RoboDK station: PintaPiezas_Dominguez_Ramirez.rdk

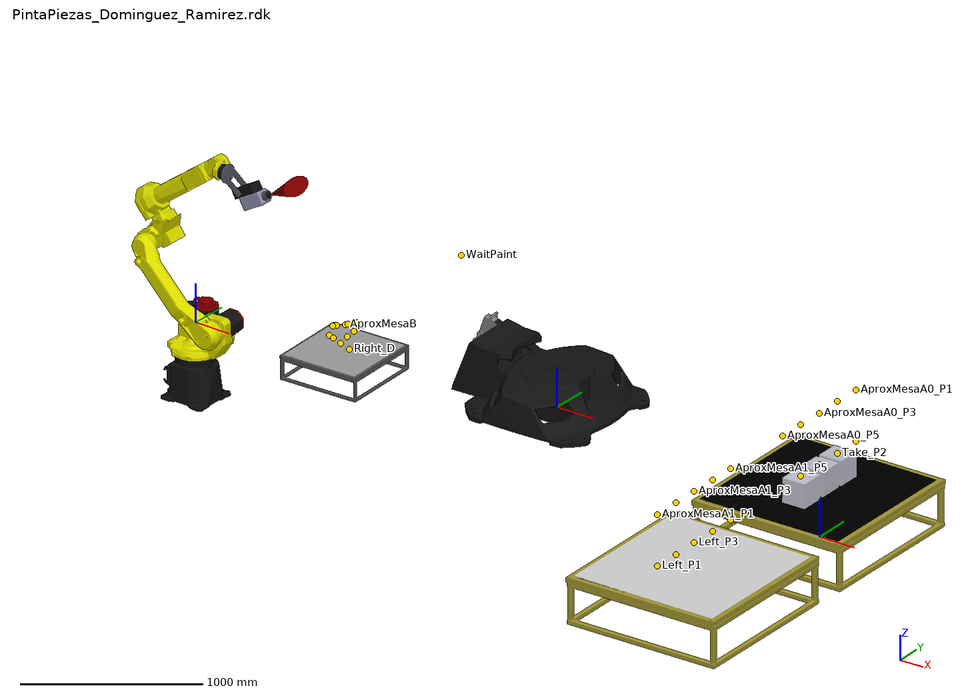
[picture v0: the station drawn from its stored meshes, robots at their saved joint values, targets as dots, program paths as lines]
Station PintaPiezas_Dominguez_Ramirez (saved by RoboDK 5.3.0). Poses are relative to the parent item; angles as X-Y-Z fixed-axis rotations.
Station parameters (name, value as stored): ColorObject, 3
  - Python program Preparar_Pieza1 (listed below)
  - Python program Pintar_Pieza1 (listed below)
  - Python program Almacenar_Pieza1 (listed below)
  - Python program Preparar_Pieza2 (listed below)
  - Python program Pintar_Pieza2 (listed below)
  - Python program Almacenar_Pieza2 (listed below)
  - Python program Preparar_Pieza3 (listed below)
  - Python program Pintar_Pieza3 (listed below)
  - Python program Almacenar_Pieza3 (listed below)
  - object MesaA at (3000, -2200, 0) mm, size 985.8 x 1004.9 x 291.9 mm, geometry from Table-108x114x32-IN.sld
    - object Pieza1 at (0, 1375, 429.65) mm, size 150 x 150 x 150 mm, geometry from box.sld
    - object Pieza2 at (0, 1200, 429.65) mm, size 150 x 150 x 150 mm, geometry from box.sld
    - object Pieza3 at (0, 1025, 429.65) mm, size 150 x 150 x 150 mm, geometry from box.sld
  - object MesaB at (0, 0, 0) mm, size 503 x 512.7 x 148.9 mm, geometry from Table-108x114x32-IN.sld
  - frame RobotA Base at (1676.97, -1606.48, 650) mm
    - robot RobotA (model KUKA KR 210 R2700 prime): 6 axes, payload 210 kg, reach 2696 mm, repeatability 0.06 mm, weight 1111 kg
        joint limits [-185, -140, -120, -350, -122.5, -350] to [185, -5, 155, 350, 122.5, 350]; home [0, -90, 90, 0, 0, 0]; saved at [-179.617, -136.253, 154.914, 0, 71.339, -179.617]
      - tool RobotiQ Sanding Kit, TCP at (0, 0, 90.86) mm, size 127 x 139.7 x 103.3 mm
    - target AproxMesaA0_P1 (Cartesian target) at (1323.03, 955.18, 93.07) mm, rotated rx 180 ry 0 rz 0 deg; joints [35.828, 52.673, -25.551, 0, -64.449, -35.828] of RobotA
    - target AproxMesaA0_P2 (Cartesian target) at (1323.03, 780.66, 93.07) mm, rotated rx 180 ry 0 rz 0 deg; joints [30.543, 46.178, -31.005, 0, -58.995, -30.543] of RobotA
    - target AproxMesaA0_P3 (Cartesian target) at (1323.03, 606.48, 93.07) mm, rotated rx -180 ry 0 rz 0 deg; joints [24.627, 41.286, -34.872, 0, -55.128, -24.627] of RobotA
    - target AproxMesaA0_P4 (Cartesian target) at (1323.03, 430.87, 93.07) mm, rotated rx -180 ry 0 rz 0 deg; joints [18.039, 37.651, -37.592, 0, -52.408, -18.039] of RobotA
    - target AproxMesaA0_P5 (Cartesian target) at (1323.03, 257.29, 93.07) mm, rotated rx -180 ry 0 rz 0 deg; joints [11.005, 35.26, -39.302, 0, -50.698, -11.005] of RobotA
    - target AproxMesaA1_P1 (Cartesian target) at (1323.03, -935.11, 93.07) mm, rotated rx -180 ry 0 rz 0 deg; joints [-35.252, 51.823, -26.284, 0, -63.716, 35.252] of RobotA
    - target AproxMesaA1_P2 (Cartesian target) at (1323.03, -761.53, 93.07) mm, rotated rx -180 ry 0 rz 0 deg; joints [-29.925, 45.572, -31.496, 0, -58.504, 29.925] of RobotA
    - target AproxMesaA1_P3 (Cartesian target) at (1323.03, -585.91, 93.07) mm, rotated rx -180 ry 0 rz 0 deg; joints [-23.886, 40.795, -35.247, 0, -54.753, 23.886] of RobotA
    - target AproxMesaA1_P4 (Cartesian target) at (1323.03, -411.74, 93.07) mm, rotated rx -180 ry 0 rz 0 deg; joints [-17.287, 37.329, -37.826, 0, -52.174, 17.287] of RobotA
    - target AproxMesaA1_P5 (Cartesian target) at (1323.03, -237.21, 93.07) mm, rotated rx -180 ry 0 rz 0 deg; joints [-10.165, 35.061, -39.441, 0, -50.559, 10.165] of RobotA
    - target Take_P1 (Cartesian target) at (1323.03, 956.48, -220.35) mm, rotated rx -180 ry 0 rz 0 deg; joints [35.865, 62.489, -38.726, 0, -51.274, -35.865] of RobotA
    - target Take_P2 (Cartesian target) at (1323.03, 780.66, -220.35) mm, rotated rx -180 ry 0 rz 0 deg; joints [30.543, 56.858, -44.792, 0, -45.208, -30.543] of RobotA
    - target Take_P3 (Cartesian target) at (1323.03, 606.48, -220.35) mm, rotated rx -180 ry 0 rz 0 deg; joints [24.627, 52.739, -49.29, 0, -40.71, -24.627] of RobotA
    - target Take_P4 (Cartesian target) at (1323.03, 430.87, -220.35) mm, rotated rx -180 ry 0 rz 0 deg; joints [18.039, 49.747, -52.598, 0, -37.402, -18.039] of RobotA
    - target Take_P5 (Cartesian target) at (1323.03, 257.29, -220.35) mm, rotated rx -180 ry 0 rz 0 deg; joints [11.005, 47.819, -54.753, 0, -35.247, -11.005] of RobotA
    - target Left_P1 (Cartesian target) at (1323.03, -933.81, -220.35) mm, rotated rx -180 ry 0 rz 0 deg; joints [-35.215, 61.659, -39.615, 0, -50.385, 35.215] of RobotA
    - target Left_P2 (Cartesian target) at (1323.03, -760.23, -220.35) mm, rotated rx -180 ry 0 rz 0 deg; joints [-29.882, 56.308, -45.389, 0, -44.611, 29.882] of RobotA
    - target Left_P3 (Cartesian target) at (1323.03, -584.61, -220.35) mm, rotated rx -180 ry 0 rz 0 deg; joints [-23.839, 52.306, -49.766, 0, -40.234, 23.839] of RobotA
    - target Left_P4 (Cartesian target) at (1323.03, -410.44, -220.35) mm, rotated rx -180 ry 0 rz 0 deg; joints [-17.235, 49.468, -52.909, 0, -37.091, 17.235] of RobotA
    - target Left_P5 (Cartesian target) at (1323.03, -235.91, -220.35) mm, rotated rx -180 ry 0 rz 0 deg; joints [-10.11, 47.649, -54.944, 0, -35.056, 10.11] of RobotA
    - target AproxMesaB (Cartesian target) at (-1417.07, 4.29, 103.23) mm, rotated rx 180 ry 0 rz 0 deg; joints [179.826, 38.777, -36.006, 0, -53.994, -179.826] of RobotA
    - target WaitPaint (Cartesian target) at (-643.02, 4.29, 741.53) mm, rotated rx 180 ry 0 rz 0 deg; joints [179.617, -20.046, -8.465, 0, -81.535, -179.617] of RobotA
    - frame MesaA0 Base at (1323.03, 606.48, -660.35) mm
      - object MesaC at (0, 0, 0) mm, size 985.8 x 1004.9 x 291.9 mm, geometry from Table-108x114x32-IN.sld
  - frame RobotB Base at (-785.52, -1535.25, 450) mm, rotated rx 0 ry 0 rz -3 deg
    - robot RobotB (model Fanuc M-10iA): 6 axes, payload 10 kg, reach 1420 mm, repeatability 0.08 mm, weight 130 kg
        modified DH rows (alpha deg, a mm, theta deg, d mm): 0, 0, 0, 450; -90, 150, -90, 0; 0, 600, 0, 0; -90, 200, 0, 640; 90, 0, 0, 0; -90, 0, 0, 100
        base shift (0, 0, -450) mm
        joint limits [-180, -90, -95, -190, -190, -360] to [180, 160, 180, 190, 190, 360]; home [0, -44.52, 36.95, 0, -36.95, 0]; saved at [0, -44.52, 36.95, 180, 36.95, 180]
      - tool Paint gun, TCP at (50, 0, 450) mm, rotated rx 0 ry 30 rz 0 deg, size 203.2 x 279.7 x 471.5 mm
    - target Right_D (Cartesian target) at (1128.46, -77.94, 203.78) mm, rotated rx 90 ry -60.18 rz -173.2 deg; joints [-28.769, 42.471, -20.584, -58.905, -97.457, 150.668] of RobotB
    - target Right_M (Cartesian target) at (1071.48, -84.74, 225.06) mm, rotated rx 90 ry -60.18 rz -173.2 deg; joints [-30.393, 36.873, -21.966, -58.048, -98.024, 152.655] of RobotB
    - target Right_U (Cartesian target) at (1002.27, -93, 254.88) mm, rotated rx 90 ry -60.18 rz -173.2 deg; joints [-32.542, 30.646, -22.514, -57, -99.408, 154.203] of RobotB
    - target Center_D (Cartesian target) at (1011.4, -39.87, 300.37) mm, rotated rx 180 ry 0 rz -173.2 deg; joints [-4.924, -0.5, 0.153, -6.683, -60.84, 193.459] of RobotB
    - target Center_M (Cartesian target) at (1050.89, 5.93, 300.37) mm, rotated rx 180 ry 0 rz -173.2 deg; joints [-1.501, 3.048, 0.227, -4.756, -60.572, 189.546] of RobotB
    - target Center_U (Cartesian target) at (1079.26, 49.09, 300.37) mm, rotated rx 180 ry 0 rz -173.2 deg; joints [1.46, 5.834, 0.429, -3.065, -60.572, 186.138] of RobotB
    - target Left_U (Cartesian target) at (1098.26, 69.52, 285.71) mm, rotated rx -90 ry 0 rz -173.2 deg; joints [33.722, 20.618, -41.647, 92.049, -87.698, 138.311] of RobotB
    - target Left_M (Cartesian target) at (1048.72, 63.61, 234.84) mm, rotated rx -90 ry 0 rz -173.2 deg; joints [35.116, 19.049, -47.063, 91.235, -88.851, 132.925] of RobotB
    - target Left_D (Cartesian target) at (1007.9, 58.74, 193.57) mm, rotated rx -90 ry 0 rz -173.2 deg; joints [36.368, 18.195, -51.506, 90.34, -89.729, 128.493] of RobotB
    - target Face_D (Cartesian target) at (972.74, -18.59, 202.79) mm, rotated rx 0 ry -90 rz -173.2 deg; joints [-9.324, -34.09, -22.694, 120.254, 16.17, 246.957] of RobotB
    - target Face_U (Cartesian target) at (973.71, -26.75, 277.71) mm, rotated rx 0 ry -90 rz -173.2 deg; joints [-10.259, -34.141, -16.259, 134.328, 20.806, 232.465] of RobotB
  - program MainProgram (9 instructions, listed below)

--- Python program Preparar_Pieza1 ---
from robolink import *    # RoboDK API
from robodk import *      # Robot toolBox
RDK = Robolink()

# Asignacion de objetos
toolA = 'RobotiQ Sanding Kit'
toolB = 'Paint gun'
objectA = 'Pieza1'
mesa1 = 'MesaB'
mesa2 = 'MesaA'
gripper1 = RDK.Item(toolA, ITEM_TYPE_TOOL)
gripper2 = RDK.Item(toolB, ITEM_TYPE_TOOL)
pi2 = RDK.Item(objectA, ITEM_TYPE_OBJECT)
mesapaint = RDK.Item(mesa1, ITEM_TYPE_OBJECT)
mesafinal = RDK.Item(mesa2, ITEM_TYPE_OBJECT)

# Configuracion RobotA
robotA = RDK.ItemUserPick('RobotA',ITEM_TYPE_ROBOT)
if not robotA.Valid():
    quit()
reference = robotA.Parent()
robotA.setPoseFrame(reference)
pose_ref = robotA.Pose()
print(Pose_2_TxyzRxyz(pose_ref))
home_joints = robotA.JointsHome().tolist()

# Preparar Pieza1 con Pick & Place

# RobotA se aproxima a MesaC para recoger la Pieza1
RDK.Spray_Clear()               # Se resetea el color de pintura
pi2.Recolor([0.90,0.91,0.96,1]) # Selecciona blanco como color inicial de la Pieza1
aprox=20
a1 = transl(1323.030,780.657,93.068)*roty(pi)
robotA.MoveJ(a1)
robotA.setSpeed(1000)

# RobotA toma la Pieza1 de la MesaC
b1 = transl(1323.030,780.657,-220.350)*roty(pi)
robotA.MoveJ(b1)
robotA.setSpeed(1000)
pi2.setParentStatic(gripper1)

# RobotA lleva la Pieza1 cerca de la MesaB
c1=transl(-1417.075,4.293,400.446)*roty(pi)
robotA.MoveJ(c1)
robotA.setSpeed(1000)

# RobotA deja la Pieza1 en la MesaB
d1=transl(-1417.075,4.293,100.367)*roty(pi)
robotA.MoveJ(d1)
robotA.setSpeed(1000)
gripper1.DetachAll()
pi2.setParentStatic(mesapaint)

# RobotA se ubica en la posición de espera
e1=transl(-643.019,4.293,741.529)*roty(pi)
robotA.MoveJ(e1)
robotA.setSpeed(1000)

--- Python program Pintar_Pieza1 ---
from robolink import *    # RoboDK API
from robodk import *      # Robot toolBox
RDK = Robolink()

# Asignacion de objetos
toolA = 'RobotiQ Sanding Kit'
toolB = 'Paint gun'
objectA = 'Pieza1'
mesa1 = 'MesaB'
mesa2 = 'MesaA'
gripper1 = RDK.Item(toolA, ITEM_TYPE_TOOL)
gripper2 = RDK.Item(toolB, ITEM_TYPE_TOOL)
pi1 = RDK.Item(objectA, ITEM_TYPE_OBJECT)
mesapaint = RDK.Item(mesa1, ITEM_TYPE_OBJECT)
mesafinal = RDK.Item(mesa2, ITEM_TYPE_OBJECT)

# Configuracion RobotB
robotB = RDK.ItemUserPick('RobotB',ITEM_TYPE_ROBOT)
if not robotB.Valid():
    quit()
reference1 = robotB.Parent()
robotB.setPoseFrame(reference1)
pose_ref1 = robotB.Pose()
print(Pose_2_TxyzRxyz(pose_ref1))
home_joints1 = robotB.JointsHome().tolist()

# RobotB pinta Pieza1
# Elegir color
color_object = 0
color_object_input = int(mbox('Seleccione un color ingresando el valor numerico correspondiente: 1=Rojo, 2=Verde, 3=Azul', entry=color_object))

# RobotB se aproxima a MesaB
aprox=20
a02 = xyzrpw_2_pose([951.091,-99.100,515.373,90.000,-60.175,-173.197])
robotB.MoveJ(a02)
robotB.setSpeed(100)

# Lado derecho
aprox=20
a2 = xyzrpw_2_pose([1128.463,-77.940,203.783,90.000,-60.175,-173.197])
robotB.MoveJ(a2)
robotB.setSpeed(100)
c2 = xyzrpw_2_pose([1071.476,-84.739,225.057,90.000,-60.175,-173.197])
robotB.MoveJ(c2)
robotB.setSpeed(1000)
d2 = xyzrpw_2_pose([1002.267,-92.996,254.878,90.000,-60.175,-173.197])
robotB.MoveJ(d2)
robotB.setSpeed(1000)

# Centro
e2 = xyzrpw_2_pose([1011.397,-39.866,300.368,180.000,0.000,-173.197])
robotB.MoveJ(e2)
robotB.setSpeed(1000)
f2 = xyzrpw_2_pose([1050.893,5.934,300.367,180.000,0.000,-173.197])
robotB.MoveJ(f2)
robotB.setSpeed(1000)
g2 = xyzrpw_2_pose([1079.262,49.092,300.367,180.000,0.000,-173.197])
robotB.MoveJ(g2)
robotB.setSpeed(1000)

# Lado izquierdo
h2 = xyzrpw_2_pose([1098.260,69.520,285.711,-90.000,0.000,-173.197])
robotB.MoveJ(h2)
robotB.setSpeed(1000)
i2 = xyzrpw_2_pose([1048.722,63.609,234.840,-90.000,0.000,-173.197])
robotB.MoveJ(i2)
robotB.setSpeed(1000)
j2 = xyzrpw_2_pose([1007.902,58.739,193.572,-90.000,0.000,-173.197])
robotB.MoveJ(j2)
robotB.setSpeed(1000)

# Frente
k2 = xyzrpw_2_pose([972.738,-18.594,202.789,0.000,-90.000,-173.197])
robotB.MoveJ(k2)
robotB.setSpeed(1000)
l2 = xyzrpw_2_pose([973.710,-26.748,277.710,0.000,-90.000,-173.197])
robotB.MoveJ(l2)
robotB.setSpeed(1000)

# Volver a la posicion inical
b2 = xyzrpw_2_pose([670.544,0.000,1022.351,0.000,-60.000,-180.000])
robotB.MoveJ(b2)
robotB.setSpeed(100)

# Color
if color_object_input == 1:
    pi1.Recolor([1,0,0,1])
elif color_object_input == 2:
    pi1.Recolor([0,1,0,1])
elif color_object_input == 3:
    pi1.Recolor([0,0,1,1])
else:
    pi1.Recolor([0.90,0.91,0.96,1])

--- Python program Almacenar_Pieza1 ---
from robolink import *    # RoboDK API
from robodk import *      # Robot toolBox
RDK = Robolink()

# Asignacion de objetos
toolA = 'RobotiQ Sanding Kit'
toolB = 'Paint gun'
objectA = 'Pieza1'
mesa1 = 'MesaB'
mesa2 = 'MesaA'
gripper1 = RDK.Item(toolA, ITEM_TYPE_TOOL)
gripper2 = RDK.Item(toolB, ITEM_TYPE_TOOL)
pi2 = RDK.Item(objectA, ITEM_TYPE_OBJECT)
mesapaint = RDK.Item(mesa2, ITEM_TYPE_OBJECT)
mesafinal = RDK.Item(mesa2, ITEM_TYPE_OBJECT)

# Configuracion RobotA
robotA = RDK.ItemUserPick('RobotA',ITEM_TYPE_ROBOT)
if not robotA.Valid():
    quit()
reference = robotA.Parent()
robotA.setPoseFrame(reference)
pose_ref = robotA.Pose()
print(Pose_2_TxyzRxyz(pose_ref))
home_joints = robotA.JointsHome().tolist()

# Almacenar Pieza1 con Pick & Place

# RobotA toma la Pieza1 de la MesaB
a3=transl(-1417.075,4.293,100.367)*roty(pi)
robotA.MoveJ(a3)
robotA.setSpeed(1000)
mesapaint.DetachAll()
pi2.setParentStatic(gripper1)

# RobotA lleva la Pieza1 lejos de la MesaB
b3=transl(-1417.075,4.293,400.446)*roty(pi)
robotA.MoveJ(b3)
robotA.setSpeed(1000)

# RobotA lleva la Pieza1 entre MesaB y MesaA
f3=transl(1323.030,780.657,93.068)*roty(pi)
robotA.MoveJ(f3)
robotA.setSpeed(1000)

# RobotA lleva la Pieza1 cerca de la MesaA
c3=transl(1323.030,-761.529,93.068)*roty(pi)
robotA.MoveJ(c3)
robotA.setSpeed(1000)

# RobotA deja la Pieza1 en la MesaA
d3=transl(1323.030,-760.228,-220.350)*roty(pi)
robotA.MoveJ(d3)
robotA.setSpeed(1000)
gripper1.DetachAll()
pi2.setParentStatic(mesafinal)

# Volver a la posicion inical
e3=transl(945.000,0.000,834.135)*roty(pi)
robotA.MoveJ(e3)
robotA.setSpeed(1000)

--- Python program Preparar_Pieza2 ---
from robolink import *    # RoboDK API
from robodk import *      # Robot toolBox
RDK = Robolink()

# Asignacion de objetos
toolA = 'RobotiQ Sanding Kit'
toolB = 'Paint gun'
objectB = 'Pieza2'
mesa1 = 'MesaB'
mesa2 = 'MesaA'
gripper1 = RDK.Item(toolA, ITEM_TYPE_TOOL)
gripper2 = RDK.Item(toolB, ITEM_TYPE_TOOL)
pi3 = RDK.Item(objectB, ITEM_TYPE_OBJECT)
mesapaint = RDK.Item(mesa1, ITEM_TYPE_OBJECT)
mesafinal = RDK.Item(mesa2, ITEM_TYPE_OBJECT)

# Configuracion RobotA
robotA = RDK.ItemUserPick('RobotA',ITEM_TYPE_ROBOT)
if not robotA.Valid():
    quit()
reference = robotA.Parent()
robotA.setPoseFrame(reference)
pose_ref = robotA.Pose()
print(Pose_2_TxyzRxyz(pose_ref))
home_joints = robotA.JointsHome().tolist()

# Preparar Pieza2 con Pick & Place

# RobotA se aproxima a MesaC para recoger la Pieza2
RDK.Spray_Clear()               # Se resetea el color de pintura
pi3.Recolor([0.90,0.91,0.96,1]) # Selecciona blanco como color inicial de la Pieza2
aprox=20
a1 = transl(1323.030,606.483,93.068)*roty(pi)
robotA.MoveJ(a1)
robotA.setSpeed(1000)

# RobotA toma la Pieza2 de la MesaC
b1 = transl(1323.030,606.483,-220.350)*roty(pi)
robotA.MoveJ(b1)
robotA.setSpeed(1000)
pi3.setParentStatic(gripper1)

# RobotA lleva la Pieza2 cerca de la MesaB
c1=transl(-1417.075,4.293,400.446)*roty(pi)
robotA.MoveJ(c1)
robotA.setSpeed(1000)

# RobotA deja la Pieza2 en la MesaB
d1=transl(-1417.075,4.293,100.367)*roty(pi)
robotA.MoveJ(d1)
robotA.setSpeed(1000)
gripper1.DetachAll()
pi3.setParentStatic(mesapaint)

# RobotA se ubica en la posición de espera
e1=transl(-643.019,4.293,741.529)*roty(pi)
robotA.MoveJ(e1)
robotA.setSpeed(1000)

--- Python program Pintar_Pieza2 ---
from robolink import *    # RoboDK API
from robodk import *      # Robot toolBox
RDK = Robolink()

# Asignacion de objetos
toolA = 'RobotiQ Sanding Kit'
toolB = 'Paint gun'
objectB = 'Pieza2'
mesa1 = 'MesaB'
mesa2 = 'MesaA'
gripper1 = RDK.Item(toolA, ITEM_TYPE_TOOL)
gripper2 = RDK.Item(toolB, ITEM_TYPE_TOOL)
pi2 = RDK.Item(objectB, ITEM_TYPE_OBJECT)
mesapaint = RDK.Item(mesa1, ITEM_TYPE_OBJECT)
mesafinal = RDK.Item(mesa2, ITEM_TYPE_OBJECT)

# Configuracion RobotB
robotB = RDK.ItemUserPick('RobotB',ITEM_TYPE_ROBOT)
if not robotB.Valid():
    quit()
reference1 = robotB.Parent()
robotB.setPoseFrame(reference1)
pose_ref1 = robotB.Pose()
print(Pose_2_TxyzRxyz(pose_ref1))
home_joints1 = robotB.JointsHome().tolist()

# RobotB pinta Pieza2
# Elegir color
color_object = 0
color_object_input = int(mbox('Seleccione un color ingresando el valor numerico correspondiente: 1=Rojo, 2=Verde, 3=Azul', entry=color_object))

# RobotB se aproxima a MesaB
aprox=20
a02 = xyzrpw_2_pose([951.091,-99.100,515.373,90.000,-60.175,-173.197])
robotB.MoveJ(a02)
robotB.setSpeed(100)

# Lado derecho
aprox=20
a2 = xyzrpw_2_pose([1128.463,-77.940,203.783,90.000,-60.175,-173.197])
robotB.MoveJ(a2)
robotB.setSpeed(100)
c2 = xyzrpw_2_pose([1071.476,-84.739,225.057,90.000,-60.175,-173.197])
robotB.MoveJ(c2)
robotB.setSpeed(1000)
d2 = xyzrpw_2_pose([1002.267,-92.996,254.878,90.000,-60.175,-173.197])
robotB.MoveJ(d2)
robotB.setSpeed(1000)

# Centro
e2 = xyzrpw_2_pose([1011.397,-39.866,300.368,180.000,0.000,-173.197])
robotB.MoveJ(e2)
robotB.setSpeed(1000)
f2 = xyzrpw_2_pose([1050.893,5.934,300.367,180.000,0.000,-173.197])
robotB.MoveJ(f2)
robotB.setSpeed(1000)
g2 = xyzrpw_2_pose([1079.262,49.092,300.367,180.000,0.000,-173.197])
robotB.MoveJ(g2)
robotB.setSpeed(1000)

# Lado izquierdo
h2 = xyzrpw_2_pose([1098.260,69.520,285.711,-90.000,0.000,-173.197])
robotB.MoveJ(h2)
robotB.setSpeed(1000)
i2 = xyzrpw_2_pose([1048.722,63.609,234.840,-90.000,0.000,-173.197])
robotB.MoveJ(i2)
robotB.setSpeed(1000)
j2 = xyzrpw_2_pose([1007.902,58.739,193.572,-90.000,0.000,-173.197])
robotB.MoveJ(j2)
robotB.setSpeed(1000)

# Frente
k2 = xyzrpw_2_pose([972.738,-18.594,202.789,0.000,-90.000,-173.197])
robotB.MoveJ(k2)
robotB.setSpeed(1000)
l2 = xyzrpw_2_pose([973.710,-26.748,277.710,0.000,-90.000,-173.197])
robotB.MoveJ(l2)
robotB.setSpeed(1000)

# Volver a la posicion inical
b2 = xyzrpw_2_pose([670.544,0.000,1022.351,0.000,-60.000,-180.000])
robotB.MoveJ(b2)
robotB.setSpeed(100)

#Color
if color_object_input == 1:
    pi2.Recolor([1,0,0,1])
elif color_object_input == 2:
    pi2.Recolor([0,1,0,1])
elif color_object_input == 3:
    pi2.Recolor([0,0,1,1])
else:
    pi2.Recolor([0.90,0.91,0.96,1])

--- Python program Almacenar_Pieza2 ---
from robolink import *    # RoboDK API
from robodk import *      # Robot toolBox
RDK = Robolink()

# Asignacion de objetos
toolA = 'RobotiQ Sanding Kit'
toolB = 'Paint gun'
objectB = 'Pieza2'
mesa1 = 'MesaB'
mesa2 = 'MesaA'
gripper1 = RDK.Item(toolA, ITEM_TYPE_TOOL)
gripper2 = RDK.Item(toolB, ITEM_TYPE_TOOL)
pi3 = RDK.Item(objectB, ITEM_TYPE_OBJECT)
mesapaint = RDK.Item(mesa2, ITEM_TYPE_OBJECT)
mesafinal = RDK.Item(mesa2, ITEM_TYPE_OBJECT)

# Configuracion RobotA
robotA = RDK.ItemUserPick('RobotA',ITEM_TYPE_ROBOT)
if not robotA.Valid():
    quit()
reference = robotA.Parent()
robotA.setPoseFrame(reference)
pose_ref = robotA.Pose()
print(Pose_2_TxyzRxyz(pose_ref))
home_joints = robotA.JointsHome().tolist()

# Almacenar Pieza2 con Pick & Place

# RobotA toma la Pieza2 de la MesaB
a3=transl(-1417.075,4.293,100.367)*roty(pi)
robotA.MoveJ(a3)
robotA.setSpeed(1000)
mesapaint.DetachAll()
pi3.setParentStatic(gripper1)

# RobotA lleva la Pieza2 lejos de la MesaB
b3=transl(-1417.075,4.293,400.446)*roty(pi)
robotA.MoveJ(b3)
robotA.setSpeed(1000)

# RobotA lleva la Pieza2 entre MesaB y MesaA
f3=transl(1323.030,606.483,93.068)*roty(pi)
robotA.MoveJ(f3)
robotA.setSpeed(1000)

# RobotA lleva la Pieza2 cerca de la MesaA
c3=transl(1323.030,-585.913,93.068)*roty(pi)
robotA.MoveJ(c3)
robotA.setSpeed(1000)

# RobotA deja la Pieza2 en la MesaA
d3=transl(1323.030,-584.612,-220.350)*roty(pi)
robotA.MoveJ(d3)
robotA.setSpeed(1000)
gripper1.DetachAll()
pi3.setParentStatic(mesafinal)

# Volver a la posicion inical
e3=transl(945.000,0.000,834.135)*roty(pi)
robotA.MoveJ(e3)
robotA.setSpeed(1000)

--- Python program Preparar_Pieza3 ---
from robolink import *    # RoboDK API
from robodk import *      # Robot toolBox
RDK = Robolink()

# Asignacion de objetos
toolA = 'RobotiQ Sanding Kit'
toolB = 'Paint gun'
objectC = 'Pieza3'
mesa1 = 'MesaB'
mesa2 = 'MesaA'
gripper1 = RDK.Item(toolA, ITEM_TYPE_TOOL)
gripper2 = RDK.Item(toolB, ITEM_TYPE_TOOL)
pi4 = RDK.Item(objectC, ITEM_TYPE_OBJECT)
mesapaint = RDK.Item(mesa1, ITEM_TYPE_OBJECT)
mesafinal = RDK.Item(mesa2, ITEM_TYPE_OBJECT)

# Configuracion RobotA
robotA = RDK.ItemUserPick('RobotA',ITEM_TYPE_ROBOT)
if not robotA.Valid():
    quit()
reference = robotA.Parent()
robotA.setPoseFrame(reference)
pose_ref = robotA.Pose()
print(Pose_2_TxyzRxyz(pose_ref))
home_joints = robotA.JointsHome().tolist()

# Preparar Pieza3 con Pick & Place

# RobotA se aproxima a MesaC para recoger la Pieza3
RDK.Spray_Clear()               # Se resetea el color de pintura
pi4.Recolor([0.90,0.91,0.96,1]) # Selecciona blanco como color inicial de la Pieza3
aprox=20
a1 = transl(1323.030,430.867,93.068)*roty(pi)
robotA.MoveJ(a1)
robotA.setSpeed(1000)

# RobotA toma la Pieza3 de la MesaC
b1 = transl(1323.030,430.867,-220.350)*roty(pi)
robotA.MoveJ(b1)
robotA.setSpeed(1000)
pi4.setParentStatic(gripper1)

# RobotA lleva la Pieza3 cerca de la MesaB
c1=transl(-1417.075,4.293,400.446)*roty(pi)
robotA.MoveJ(c1)
robotA.setSpeed(1000)

# RobotA deja la Pieza3 en la MesaB
d1=transl(-1417.075,4.293,100.367)*roty(pi)
robotA.MoveJ(d1)
robotA.setSpeed(1000)
gripper1.DetachAll()
pi4.setParentStatic(mesapaint)

# RobotA se ubica en la posición de espera
e1=transl(-643.019,4.293,741.529)*roty(pi)
robotA.MoveJ(e1)
robotA.setSpeed(1000)

--- Python program Pintar_Pieza3 ---
from robolink import *    # RoboDK API
from robodk import *      # Robot toolBox
RDK = Robolink()

# Asignacion de objetos
toolA = 'RobotiQ Sanding Kit'
toolB = 'Paint gun'
objectC = 'Pieza3'
mesa1 = 'MesaB'
mesa2 = 'MesaA'
gripper1 = RDK.Item(toolA, ITEM_TYPE_TOOL)
gripper2 = RDK.Item(toolB, ITEM_TYPE_TOOL)
pi3 = RDK.Item(objectC, ITEM_TYPE_OBJECT)
mesapaint = RDK.Item(mesa1, ITEM_TYPE_OBJECT)
mesafinal = RDK.Item(mesa2, ITEM_TYPE_OBJECT)

# Configuracion RobotB
robotB = RDK.ItemUserPick('RobotB',ITEM_TYPE_ROBOT)
if not robotB.Valid():
    quit()
reference1 = robotB.Parent()
robotB.setPoseFrame(reference1)
pose_ref1 = robotB.Pose()
print(Pose_2_TxyzRxyz(pose_ref1))
home_joints1 = robotB.JointsHome().tolist()

# RobotB pinta Pieza3
# Elegir color
color_object = 0
color_object_input = int(mbox('Seleccione un color ingresando el valor numerico correspondiente: 1=Rojo, 2=Verde, 3=Azul', entry=color_object))

# RobotB se aproxima a MesaB
aprox=20
a02 = xyzrpw_2_pose([951.091,-99.100,515.373,90.000,-60.175,-173.197])
robotB.MoveJ(a02)
robotB.setSpeed(100)

# Lado derecho
aprox=20
a2 = xyzrpw_2_pose([1128.463,-77.940,203.783,90.000,-60.175,-173.197])
robotB.MoveJ(a2)
robotB.setSpeed(100)
c2 = xyzrpw_2_pose([1071.476,-84.739,225.057,90.000,-60.175,-173.197])
robotB.MoveJ(c2)
robotB.setSpeed(1000)
d2 = xyzrpw_2_pose([1002.267,-92.996,254.878,90.000,-60.175,-173.197])
robotB.MoveJ(d2)
robotB.setSpeed(1000)

# Centro
e2 = xyzrpw_2_pose([1011.397,-39.866,300.368,180.000,0.000,-173.197])
robotB.MoveJ(e2)
robotB.setSpeed(1000)
f2 = xyzrpw_2_pose([1050.893,5.934,300.367,180.000,0.000,-173.197])
robotB.MoveJ(f2)
robotB.setSpeed(1000)
g2 = xyzrpw_2_pose([1079.262,49.092,300.367,180.000,0.000,-173.197])
robotB.MoveJ(g2)
robotB.setSpeed(1000)

# Lado izquierdo
h2 = xyzrpw_2_pose([1098.260,69.520,285.711,-90.000,0.000,-173.197])
robotB.MoveJ(h2)
robotB.setSpeed(1000)
i2 = xyzrpw_2_pose([1048.722,63.609,234.840,-90.000,0.000,-173.197])
robotB.MoveJ(i2)
robotB.setSpeed(1000)
j2 = xyzrpw_2_pose([1007.902,58.739,193.572,-90.000,0.000,-173.197])
robotB.MoveJ(j2)
robotB.setSpeed(1000)

# Frente
k2 = xyzrpw_2_pose([972.738,-18.594,202.789,0.000,-90.000,-173.197])
robotB.MoveJ(k2)
robotB.setSpeed(1000)
l2 = xyzrpw_2_pose([973.710,-26.748,277.710,0.000,-90.000,-173.197])
robotB.MoveJ(l2)
robotB.setSpeed(1000)

# Volver a la posicion inical
b2 = xyzrpw_2_pose([670.544,0.000,1022.351,0.000,-60.000,-180.000])
robotB.MoveJ(b2)
robotB.setSpeed(100)

#Color
if color_object_input == 1:
    pi3.Recolor([1,0,0,1])
elif color_object_input == 2:
    pi3.Recolor([0,1,0,1])
elif color_object_input == 3:
    pi3.Recolor([0,0,1,1])
else:
    pi3.Recolor([0.90,0.91,0.96,1])

--- Python program Almacenar_Pieza3 ---
from robolink import *    # RoboDK API
from robodk import *      # Robot toolBox
RDK = Robolink()

# Asignacion de objetos
toolA = 'RobotiQ Sanding Kit'
toolB = 'Paint gun'
objectC = 'Pieza3'
mesa1 = 'MesaB'
mesa2 = 'MesaA'
gripper1 = RDK.Item(toolA, ITEM_TYPE_TOOL)
gripper2 = RDK.Item(toolB, ITEM_TYPE_TOOL)
pi4 = RDK.Item(objectC, ITEM_TYPE_OBJECT)
mesapaint = RDK.Item(mesa2, ITEM_TYPE_OBJECT)
mesafinal = RDK.Item(mesa2, ITEM_TYPE_OBJECT)

# Configuracion RobotA
robotA = RDK.ItemUserPick('RobotA',ITEM_TYPE_ROBOT)
if not robotA.Valid():
    quit()
reference = robotA.Parent()
robotA.setPoseFrame(reference)
pose_ref = robotA.Pose()
print(Pose_2_TxyzRxyz(pose_ref))
home_joints = robotA.JointsHome().tolist()

# Almacenar Pieza3 con Pick & Place

# RobotA toma la Pieza3 de la MesaB
a3=transl(-1417.075,4.293,100.367)*roty(pi)
robotA.MoveJ(a3)
robotA.setSpeed(1000)
mesapaint.DetachAll()
pi4.setParentStatic(gripper1)

# RobotA lleva la Pieza3 lejos de la MesaB
b3=transl(-1417.075,4.293,400.446)*roty(pi)
robotA.MoveJ(b3)
robotA.setSpeed(1000)

# RobotA lleva la Pieza3 entre MesaB y MesaA
f3=transl(1323.030,430.867,93.068)*roty(pi)
robotA.MoveJ(f3)
robotA.setSpeed(1000)

# RobotA lleva la Pieza3 cerca de la MesaA
c3=transl(1323.030,-411.739,93.068)*roty(pi)
robotA.MoveJ(c3)
robotA.setSpeed(1000)

# RobotA deja la Pieza3 en la MesaA
d3=transl(1323.030,-410.438,-220.350)*roty(pi)
robotA.MoveJ(d3)
robotA.setSpeed(1000)
gripper1.DetachAll()
pi4.setParentStatic(mesafinal)

# Volver a la posicion inical
e3=transl(945.000,0.000,834.135)*roty(pi)
robotA.MoveJ(e3)
robotA.setSpeed(1000)

--- program MainProgram (robot RobotA) ---
  Call Preparar_Pieza1
  Call Pintar_Pieza1
  Call Almacenar_Pieza1
  Call Preparar_Pieza2
  Call Pintar_Pieza2
  Call Almacenar_Pieza2
  Call Preparar_Pieza3
  Call Pintar_Pieza3
  Call Almacenar_Pieza3
